// TIA Portal V17 export
// export: Created 2025-06-25T13:13:09.4466625Z, ExportSetting WithDefaults, DisplayName Totally Integrated Automation Portal, DisplayVersion V17 Update 8, DisplayName TIA Portal Openness, DisplayVersion V17 Update 8, DisplayName TIA Portal Version Control Interface, DisplayVersion V17, DisplayName STEP 7 Professional, DisplayVersion V17 Update 8, DisplayName STEP 7 Safety, DisplayVersion V17 Update 6, DisplayName WinCC Advanced, DisplayVersion V17 Update 8
FUNCTION_BLOCK "Calculations"   // FB42, FBD
{ S7_Optimized_Access := 'TRUE' }
VERSION : 0.1
// stored: AutoNumber true, IsIECCheckEnabled false, IsRetainMemResEnabled false, MemoryReserve 0, SetENOAutomatically false, UDAEnableTagReadback false
   VAR
      OperatingTimeCounters_Instance { ExternalAccessible := 'False'; ExternalVisible := 'False'; ExternalWritable := 'False'; S7_SetPoint := 'True'} : "OperatingTimeCounters";
      DT1_Merker_intern { ExternalAccessible := 'False'; ExternalVisible := 'False'; ExternalWritable := 'False'; S7_SetPoint := 'True'} : Real;
   END_VAR
   VAR_TEMP
      HeatRateSource : Real;
      HeatRateSink : Real;
      COP_max : Real;
      Quality : Real;
      COP : Real;
      HeatSourceDegreesPerSec : Real;
      HeatSourceDegreesPerMin : Real;
   END_VAR
   VAR_TEMP   // added for the SCL form of the ladder/FBD networks
      _w1 : Bool;
   END_VAR
BEGIN

REGION Network 1: Compressor calculations
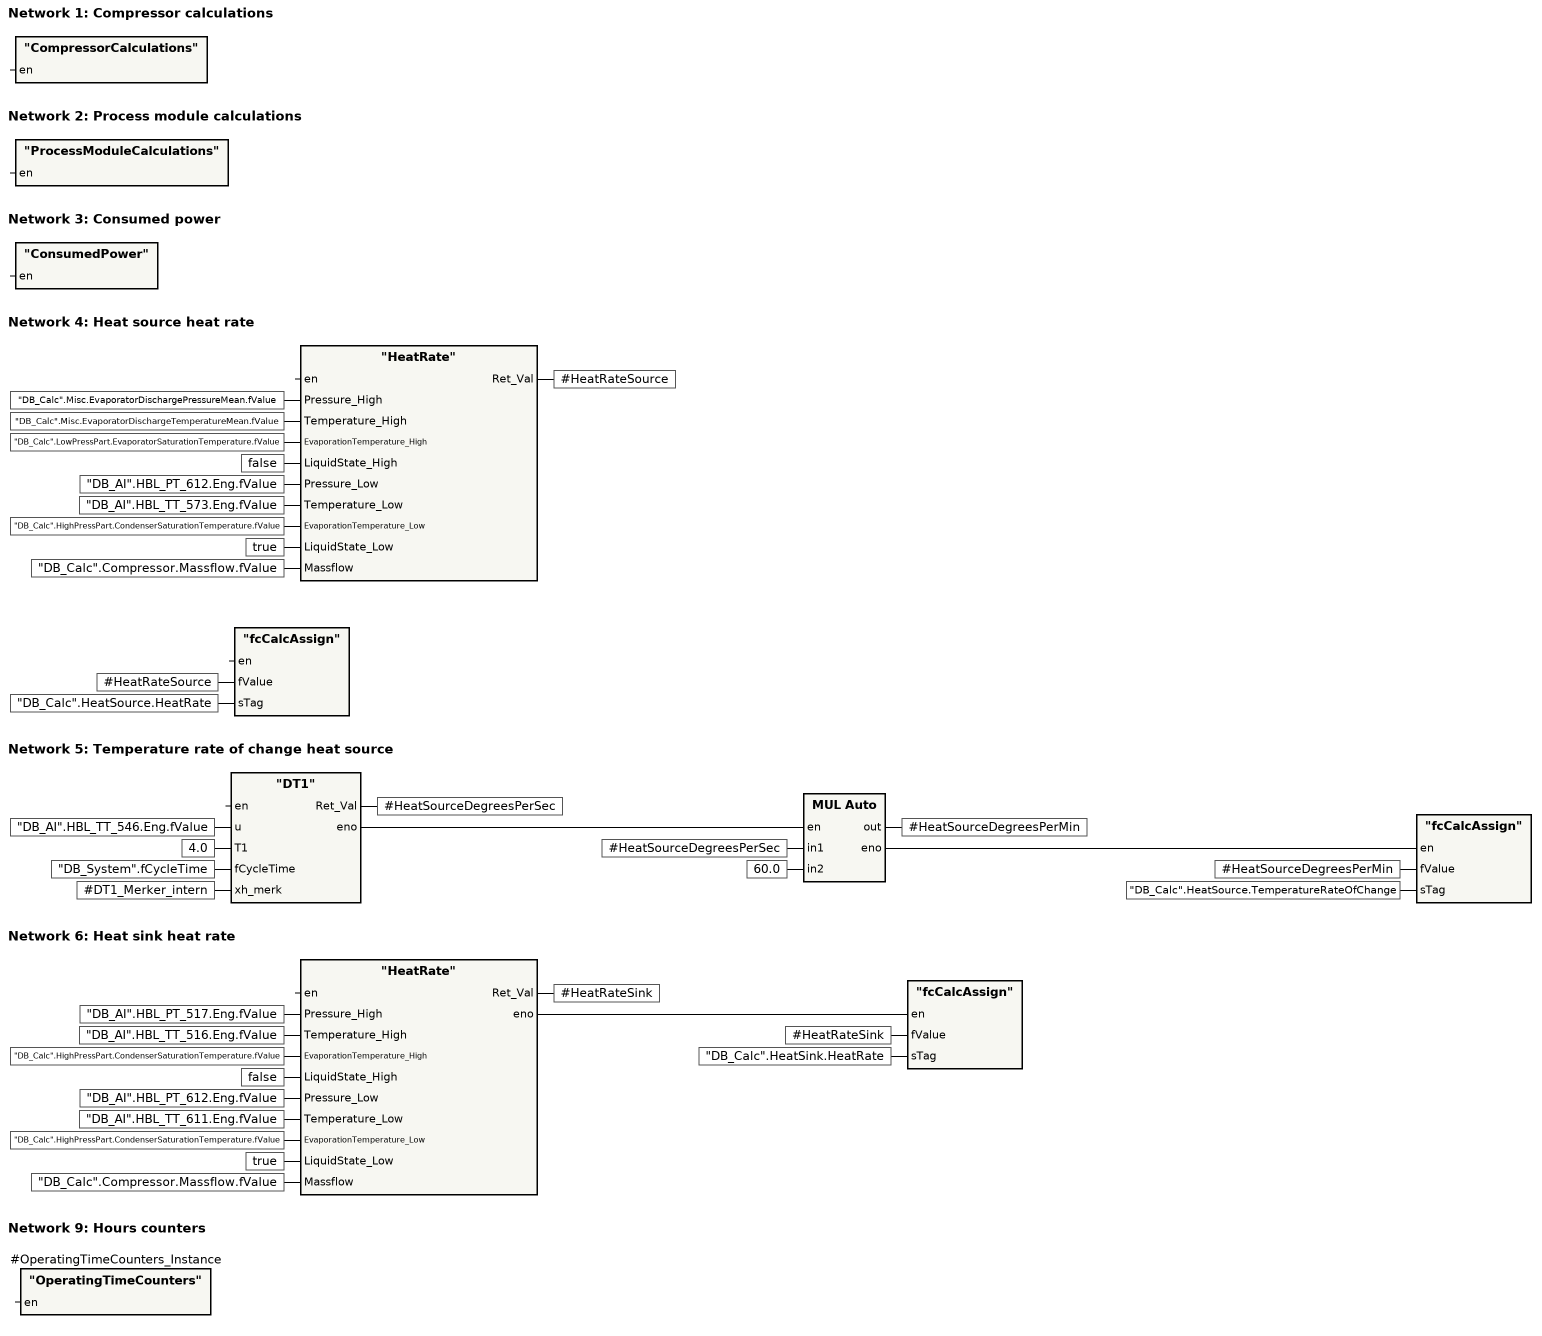
   "CompressorCalculations"();
END_REGION

REGION Network 2: Process module calculations
   "ProcessModuleCalculations"();
END_REGION

REGION Network 3: Consumed power
   "ConsumedPower"();
END_REGION

REGION Network 4: Heat source heat rate
   // The high side is the evaporator discharge temp & pressure, in gas phase
   // The low side, should be the evaporator suction temp & pressure, in liquid phase, but:
   //  - the condenser discharge pressure is used as it is the only pressure reading in that part of the system.
   //  - the expansion valve temperature is used
   // "We use the entalpy of the liquid before the expansion valve instead of the one before the evaporator, because the pressure and quality of the fluid before the evaporator is uncertain,  but it is known before the expansion valve and the expansion valve itself does not alter the enthalpy very much. "
   #HeatRateSource := "HeatRate"(Pressure_High := "DB_Calc".Misc.EvaporatorDischargePressureMean.fValue,
                           Temperature_High := "DB_Calc".Misc.EvaporatorDischargeTemperatureMean.fValue,
                           EvaporationTemperature_High := "DB_Calc".LowPressPart.EvaporatorSaturationTemperature.fValue,
                           LiquidState_High := false,
                           Pressure_Low := "DB_AI".HBL_PT_612.Eng.fValue,
                           Temperature_Low := "DB_AI".HBL_TT_573.Eng.fValue,
                           EvaporationTemperature_Low := "DB_Calc".HighPressPart.CondenserSaturationTemperature.fValue,
                           LiquidState_Low := true,
                           Massflow := "DB_Calc".Compressor.Massflow.fValue);
   "fcCalcAssign"(fValue := #HeatRateSource, sTag := "DB_Calc".HeatSource.HeatRate);
END_REGION

REGION Network 5: Temperature rate of change heat source
   // ###BE AWARE changed from K/sec to K/min
   #HeatSourceDegreesPerSec := "DT1"(u := "DB_AI".HBL_TT_546.Eng.fValue,
                           T1 := 4.0,
                           fCycleTime := "DB_System".fCycleTime,
                           xh_merk := #DT1_Merker_intern,
                           ENO => #_w1);
   IF #_w1 THEN
       #HeatSourceDegreesPerMin := #HeatSourceDegreesPerSec * 60.0;
       "fcCalcAssign"(fValue := #HeatSourceDegreesPerMin, sTag := "DB_Calc".HeatSource.TemperatureRateOfChange);
   END_IF;
END_REGION

REGION Network 6: Heat sink heat rate
   // The high side is the condenser suction temp & pressure, in gas phase
   // The low side is the condenser discharge temp & pressure, in liquid phase
   #HeatRateSink := "HeatRate"(Pressure_High := "DB_AI".HBL_PT_517.Eng.fValue,
                           Temperature_High := "DB_AI".HBL_TT_516.Eng.fValue,
                           EvaporationTemperature_High := "DB_Calc".HighPressPart.CondenserSaturationTemperature.fValue,
                           LiquidState_High := false,
                           Pressure_Low := "DB_AI".HBL_PT_612.Eng.fValue,
                           Temperature_Low := "DB_AI".HBL_TT_611.Eng.fValue,
                           EvaporationTemperature_Low := "DB_Calc".HighPressPart.CondenserSaturationTemperature.fValue,
                           LiquidState_Low := true,
                           Massflow := "DB_Calc".Compressor.Massflow.fValue,
                           ENO => #_w1);
   IF #_w1 THEN "fcCalcAssign"(fValue := #HeatRateSink, sTag := "DB_Calc".HeatSink.HeatRate); END_IF;
END_REGION

REGION Network 7 (SCL): COP
    IF "DB_Calc".System.ElectricalPower.fValue > 0.0 THEN
       #COP := "DB_Calc".HeatSink.HeatRate.fValue / "DB_Calc".System.ElectricalPower.fValue;
   ELSE
       #COP := 0.0;
   END_IF;

   "fcCalcAssign"(fValue := #COP, sTag := "DB_Calc".System.COP);
END_REGION

REGION Network 8 (SCL): Carnot quality
   // Quality rating is COP divided by COP_max (Carnot)
   // Verify this expression
   #COP_max := (("DB_AI".HBL_TT_901.Eng.fValue + "DB_AI".HBL_TT_518.Eng.fValue/2+273.15) * 
                ("DB_AI".HBL_TT_901.Eng.fValue + "DB_AI".HBL_TT_518.Eng.fValue -
                 "DB_AI".HBL_TT_542.Eng.fValue - "DB_AI".HBL_TT_546.Eng.fValue)/2 *100.0);

   IF "DB_AI".HBL_TT_542.Eng.fValue < "DB_AI".HBL_TT_901.Eng.fValue THEN
       #Quality := #COP / #COP_max;
   ELSE
       #Quality := 0.0;
   END_IF;

   "fcCalcAssign"(fValue := #Quality, sTag := "DB_Calc".System.Quality);
END_REGION

REGION Network 9: Hours counters
   #OperatingTimeCounters_Instance();   // "OperatingTimeCounters"
END_REGION

REGION Network 10: Temperature Lift
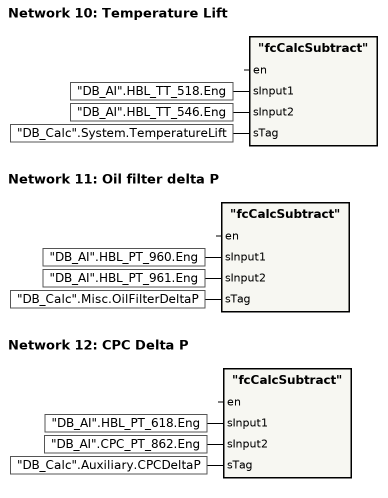
   "fcCalcSubtract"(sInput1 := "DB_AI".HBL_TT_518.Eng,
                    sInput2 := "DB_AI".HBL_TT_546.Eng,
                    sTag := "DB_Calc".System.TemperatureLift);
END_REGION

REGION Network 11: Oil filter delta P
   "fcCalcSubtract"(sInput1 := "DB_AI".HBL_PT_960.Eng,
                    sInput2 := "DB_AI".HBL_PT_961.Eng,
                    sTag := "DB_Calc".Misc.OilFilterDeltaP);
END_REGION

REGION Network 12: CPC Delta P
   // Actually the delta P over "orifice" V-861
   "fcCalcSubtract"(sInput1 := "DB_AI".HBL_PT_618.Eng,
                    sInput2 := "DB_AI".CPC_PT_862.Eng,
                    sTag := "DB_Calc".Auxiliary.CPCDeltaP);
END_REGION
END_FUNCTION_BLOCK
